FUNCTION UDINT_TO_SIZE : ST_SIZE
VAR_INPUT
	nValue : UDINT;
END_VAR

UDINT_TO_SIZE.nValue := nValue;

END_FUNCTION

(* stored: Version 1.1.0.1, ProductVersion 3.1.4024.15
   POU UDINT_TO_SIZE: Id {b65a5d58-2b30-41bf-b54e-292bc4b7f4b4}, SpecialFunc None *)
